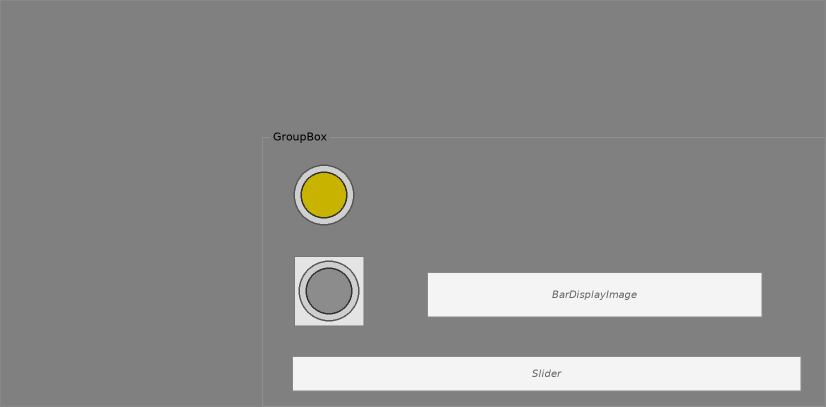
VISUALIZATION SimulatorExampleVisu  // 826x407
    GroupBox (262,129 564x278), "GroupBox"
        Lamp1 (27,31 70x70), variable: P_SimulatorExample.stWaterTankStates.bSimulatorRunning, style: Lamp-Lamp1-Yellow
        PushSwitch (32,127 70x70), variable: P_SimulatorExample.stWaterTankStates.bSimulatorRunning, behaviour: TOGGLE, style: Switch-PushSwitch-Gray
        Slider (30,227 509x35), variable: P_SimulatorExample.stWaterTankStates.fFlowIn, scale 0..10
        BarDisplayImage (165,143 335x45), value: P_SimulatorExample.stWaterTankStates.fWaterHeight, invisible if: P_SimulatorExample.stWaterTankStates.fWaterHeight, style: BarDisplayImage-Gray, scale format: %.1f, scale 0..100
END_VISUALIZATION

(* stored: Version 1.1.0.1, ProductVersion 3.1.4024.12
   Visu SimulatorExampleVisu: Id {39a9648c-c846-4fba-b98a-a173e4f9e8d3} *)
